// TwinCAT 3 PLC project InventoryManagement
// ProgramVersion: 3.1.4026.19
// libraries:
//   Tc2_Standard, * (Beckhoff Automation GmbH)
//   Tc2_System, * (Beckhoff Automation GmbH)
// project tree:
//   DUTs/ ST_Space.TcDUT
//   / PlcTask.TcTTO
//   POUs/ FB_QueueLogic.TcPOU, FB_Robot.TcPOU, FB_ShelfManager.TcPOU, InventoryManagement.TcCD (not stored), MAIN.TcPOU
// real-time tasks:
//   TASK PlcTask: cycle T#10ms, priority 20, ADS port 350

CONFIGURATION InventoryManagement
    RESOURCE PLC ON TwinCAT3
        TASK PlcTask(INTERVAL := T#10ms, PRIORITY := 20);
        PROGRAM MAIN WITH PlcTask : MAIN;
    END_RESOURCE
END_CONFIGURATION

// ---- DUTs/ST_Space.TcDUT
TYPE ST_Space :
STRUCT
	bIsOccupied		: BOOL;
	sPartID			: STRING(23);
END_STRUCT
END_TYPE

// ---- POUs/MAIN.TcPOU
PROGRAM MAIN
VAR
	fbShelf 	: FB_ShelfManager;
	fbRobot 		: FB_Robot;

    step : INT := 0;

    partID1 : STRING(23) := 'PART1_0000000000000000';
    partID2 : STRING(23) := 'PART2_0000000000000000';
    partID3 : STRING(23) := 'PART3_0000000000000000';

    pos     : INT;
    ok      : BOOL;
    outID   : STRING(23);
END_VAR

CASE step OF

    0:  
        fbShelf.LoadNextFreeSpace(
            PartID   := partID1,
            Pos      => pos,
            bSuccessful => ok
        );
        IF ok THEN step := 1; END_IF

    1:  
        fbShelf.LoadNextFreeSpace(
            PartID   := partID2,
            Pos      => pos,
            bSuccessful => ok
        );
        IF ok THEN step := 2; END_IF

    2:  
        fbShelf.LoadNextFreeSpace(
            PartID   := partID3,
            Pos      => pos,
            bSuccessful => ok
        );
        IF ok THEN step := 3; END_IF

    3:  
        fbShelf.GetNextOccupiedSpace(
            Pos      => pos,
            bSuccessful => ok
        ); 
        step := 4;

    4:  
        fbShelf.UnloadNextOccupiedSpace(
            PartID   => outID,
            Pos      => pos,
            bSuccessful => ok
        );
        step := 5;

    5:  
        fbShelf.UnloadByPartID(
            PartID   := partID2,
            Pos      => pos,
            bSuccessful => ok
        );
        step := 6;

    6: 
        fbShelf.UnloadNextOccupiedSpace(
            PartID   => outID,
            Pos      => pos,
            bSuccessful => ok
        );
        step := 100;

    100:
        step := 100;

END_CASE

END_PROGRAM

// ---- POUs/FB_ShelfManager.TcPOU
FUNCTION_BLOCK FB_ShelfManager
VAR_INPUT
END_VAR
VAR_OUTPUT
END_VAR
VAR
	aSpaces		: ARRAY [1..42] OF ST_Space;
	oQueueLogic : FB_QueueLogic;

END_VAR

METHOD GetNextFreeSpace : BOOL
VAR_INPUT
END_VAR
VAR_OUTPUT
	Pos 			: INT;
	bSuccessful		: BOOL;
END_VAR
VAR
    i : INT;
END_VAR
FOR i := 1 TO 42 DO
    IF NOT aSpaces[i].bIsOccupied THEN
        Pos := i;
        bSuccessful := TRUE;
        RETURN;
    END_IF
END_FOR

Pos := 0;
bSuccessful := FALSE;
END_METHOD

METHOD GetNextOccupiedSpace : BOOL
VAR_INPUT
END_VAR
VAR_OUTPUT
	Pos 			: INT;
	bSuccessful		: BOOL;
END_VAR
oQueueLogic.CurrentPointerPosition(iIndex => Pos,bSuccessful => bSuccessful);

IF NOT bSuccessful THEN
    Pos := 0;
END_IF
END_METHOD

METHOD GetSpaceByPartID : BOOL
VAR_INPUT
	PartID			: STRING(23);
END_VAR
VAR_OUTPUT
	Pos 			: INT;
	bSuccessful		: BOOL;
END_VAR
END_METHOD

METHOD LoadByExplicitPosition 
VAR_INPUT
	PartID : STRING(23);
	Pos : INT;
END_VAR
VAR_OUTPUT
	bSuccessful		: BOOL;
END_VAR
VAR
    bRemoved : BOOL;
END_VAR

IF (Pos < 1) OR (Pos > 42) THEN
    bSuccessful := FALSE;
    RETURN;
END_IF

IF aSpaces[Pos].bIsOccupied THEN
    oQueueLogic.RemoveByIndex(
        iIndex      := Pos,
        bSuccessful => bRemoved
    );
	IF NOT bRemoved THEN
		bSuccessful := FALSE;
        RETURN;
	END_IF
END_IF

aSpaces[Pos].bIsOccupied := TRUE;
aSpaces[Pos].sPartID := PartID;

oQueueLogic.Push(Pos);

bSuccessful := TRUE;
END_METHOD

METHOD LoadNextFreeSpace
VAR_INPUT
	PartID : STRING(23);
END_VAR
VAR_OUTPUT
    Pos : INT;
    bSuccessful : BOOL;
END_VAR
VAR
    i : INT;
END_VAR
FOR i := 1 TO 42 DO
    IF NOT aSpaces[i].bIsOccupied THEN

        aSpaces[i].bIsOccupied := TRUE;
        aSpaces[i].sPartID := PartID;

        oQueueLogic.Push(i);

        Pos := i;
        bSuccessful := TRUE;
        RETURN;
    END_IF
END_FOR

Pos := 0;
bSuccessful := FALSE;
END_METHOD

METHOD UnloadByExplicitPosition : BOOL
VAR_INPUT
	Pos : INT;
END_VAR
VAR_OUTPUT
	bSuccessful		: BOOL;
END_VAR
VAR
    bRemoved : BOOL;
END_VAR
IF (Pos < 1) OR (Pos > 42) THEN
    bSuccessful := FALSE;
    RETURN;
END_IF

IF NOT aSpaces[Pos].bIsOccupied THEN
    bSuccessful := FALSE;
    RETURN;
END_IF
oQueueLogic.RemoveByIndex(
    iIndex      := Pos,
    bSuccessful => bRemoved
);

IF NOT bRemoved THEN
    bSuccessful := FALSE;
    RETURN;
END_IF

aSpaces[Pos].bIsOccupied := FALSE;
aSpaces[Pos].sPartID := '';

bSuccessful := TRUE;
END_METHOD

METHOD UnloadByPartID : BOOL
VAR_INPUT
	PartID			: STRING(23);
END_VAR
VAR_OUTPUT
	Pos 			: INT;
	bSuccessful		: BOOL;
END_VAR
VAR
    i : INT;
    bRemoved : BOOL;
END_VAR
FOR i := 1 TO 42 DO
    IF aSpaces[i].bIsOccupied AND (aSpaces[i].sPartID = PartID) THEN

        aSpaces[i].bIsOccupied := FALSE;
        aSpaces[i].sPartID := '';

        oQueueLogic.RemoveByIndex(i, bSuccessful => bRemoved);

        Pos := i;
        bSuccessful := TRUE;
        RETURN;
    END_IF
END_FOR

Pos := 0;
bSuccessful := FALSE;
END_METHOD

METHOD UnloadNextOccupiedSpace 
VAR_INPUT
END_VAR
VAR_OUTPUT
	PartID			: STRING(23);
	Pos 			: INT;
	bSuccessful		: BOOL;
END_VAR
VAR
    iPos : INT;
END_VAR
oQueueLogic.Pop(iIndex => iPos, bSuccessful => bSuccessful);

IF NOT bSuccessful THEN
    Pos := 0;
    PartID := '';
    RETURN;
END_IF

PartID := aSpaces[iPos].sPartID;
aSpaces[iPos].bIsOccupied := FALSE;
aSpaces[iPos].sPartID := '';

Pos := iPos;
bSuccessful := TRUE;
END_METHOD

END_FUNCTION_BLOCK

// ---- POUs/FB_QueueLogic.TcPOU
FUNCTION_BLOCK FB_QueueLogic
VAR_INPUT
END_VAR
VAR_OUTPUT
END_VAR
VAR
	aQueue			: ARRAY [1..42] OF INT;
	iStartPointer	: INT;
	iEndPointer		: INT;
	nCounter		: INT := 0;
END_VAR

METHOD CurrentPointerPosition : BOOL
VAR_INPUT
END_VAR
VAR_OUTPUT
	iIndex		: INT;
	bSuccessful	: BOOL;
END_VAR

IF nCounter = 0 THEN
    bSuccessful := FALSE;
    iIndex := 0;
    RETURN;
END_IF


iIndex := aQueue[iStartPointer];
bSuccessful := TRUE;
END_METHOD

METHOD IsEmpty : BOOL
VAR_INPUT
END_VAR
VAR_OUTPUT
	bEmpty		: BOOL;
END_VAR
bEmpty := nCounter = 0;
END_METHOD

METHOD IsFull : BOOL
VAR_INPUT
END_VAR
VAR_OUTPUT
	bFull		: BOOL;
END_VAR
bFull := nCounter >= 42;
END_METHOD

METHOD Pop : BOOL
VAR_INPUT
	
END_VAR
VAR_OUTPUT
	iIndex	: INT;
	bSuccessful		: BOOL;
END_VAR

IF nCounter = 0 THEN
    bSuccessful := FALSE;
    iIndex := 0;
    RETURN;
END_IF

iIndex := aQueue[iStartPointer];
nCounter := nCounter - 1;

IF nCounter = 0 THEN   
    iStartPointer := 0;
    iEndPointer   := 0;
ELSE
    iStartPointer := iStartPointer + 1;
    IF iStartPointer > 42 THEN
        iStartPointer := 1;
    END_IF
END_IF

bSuccessful := TRUE;
END_METHOD

METHOD Push : BOOL
VAR_INPUT
	iIndex	: INT;
END_VAR
VAR_OUTPUT
	bSuccessful		: BOOL;
END_VAR
VAR
// 	i		: INT := 1;
END_VAR
// Adding the part in the Queue, increasing the nCounter and updating the Queue's Index

IF nCounter >= 42 THEN
	bSuccessful := FALSE;
	RETURN;
END_IF
IF nCounter = 0 THEN
	iStartPointer 		:= 1;
	iEndPointer   		:= 1;
ELSE
	iEndPointer := iEndPointer + 1;
	IF iEndPointer > 42 THEN
		iEndPointer := 1; 
	END_IF
END_IF
aQueue[iEndPointer] := iIndex;
	
nCounter	:=nCounter+1;
bSuccessful := TRUE;	

RETURN;
END_METHOD

METHOD RemoveByIndex : BOOL
VAR_INPUT
	iIndex	: INT;
END_VAR
VAR_OUTPUT
	bSuccessful		: BOOL;
END_VAR
VAR
	i,j,iPos		: INT;
	bFound	: BOOL;
END_VAR
IF nCounter = 0 THEN
    bSuccessful := FALSE;
    RETURN;
END_IF

iPos := iStartPointer;
bFound := FALSE;

FOR i := 1 TO nCounter DO
    IF aQueue[iPos] = iIndex THEN
        bFound := TRUE;
        EXIT;
    END_IF

    iPos := iPos + 1;
    IF iPos > 42 THEN
        iPos := 1;
    END_IF
END_FOR

IF NOT bFound THEN
    bSuccessful := FALSE;
    RETURN;
END_IF


j := iPos;
WHILE j <> iEndPointer DO
    IF j = 42 THEN
        aQueue[j] := aQueue[1];
        j := 1;
    ELSE
        aQueue[j] := aQueue[j + 1];
        j := j + 1;
    END_IF
END_WHILE


IF iEndPointer = 1 THEN
    iEndPointer := 42;
ELSE
    iEndPointer := iEndPointer - 1;
END_IF

nCounter := nCounter - 1;

(* Queue became empty *)
IF nCounter = 0 THEN
    iStartPointer := 0;
    iEndPointer := 0;
END_IF

bSuccessful := TRUE;
END_METHOD

END_FUNCTION_BLOCK

// ---- POUs/FB_Robot.TcPOU
FUNCTION_BLOCK FB_Robot
VAR_INPUT
END_VAR
VAR_OUTPUT
END_VAR
VAR
	fbShelfManager	: REFERENCE TO FB_ShelfManager;
END_VAR

METHOD LoadPart : BOOL
VAR_INPUT
	PartID : STRING(23);
END_VAR
VAR_OUTPUT
	Pos 			: INT;
	bSuccessful		: BOOL;
END_VAR
END_METHOD

METHOD UnloadPart : BOOL
VAR_INPUT
END_VAR
VAR_OUTPUT
	PartID 			: STRING(23);	
	Pos 			: INT;
	bSuccessful		: BOOL;
END_VAR
END_METHOD

END_FUNCTION_BLOCK
